{attribute addProperty BoxType "EK1100-0000-0018"}
{attribute addProperty Id "Beckhoff_APS1xxxEK1122Beckhoff_APS1xxxEK1122_85E711A32114264.25A_0002_APS1003_5000_0016APS1003_59AFCAF52546318.25"}
{attribute addProperty CRC "72743123"}
{attribute addProperty SizeInBites "4660"}
{attribute addProperty SizeInBytes "582.5"}
TYPE Beckhoff_APS1xxx_0455F8D3 EXTENDS EK1100_179A0949 :
STRUCT
	{attribute addProperty Name "Beckhoff_APS1xxxEK1122"}
	Beckhoff_APS1xxxEK1122 : Beckhoff_APS1xxxEK1122_85E711A3;
	{attribute addProperty Name "A_0002_APS1003_5000_0016"}
	A_0002_APS1003_5000_0016 : APS1003_59AFCAF5;
END_STRUCT
END_TYPE

(* stored: Version 1.2.0.0, ProductVersion 3.1.4024.9
   DUT Beckhoff_APS1xxx_0455F8D3: Id {52d742a8-8a88-4c91-95b5-650e846593b9} *)
